RoboDK station: ALTERNATIVA 3 - PYTHON.rdk

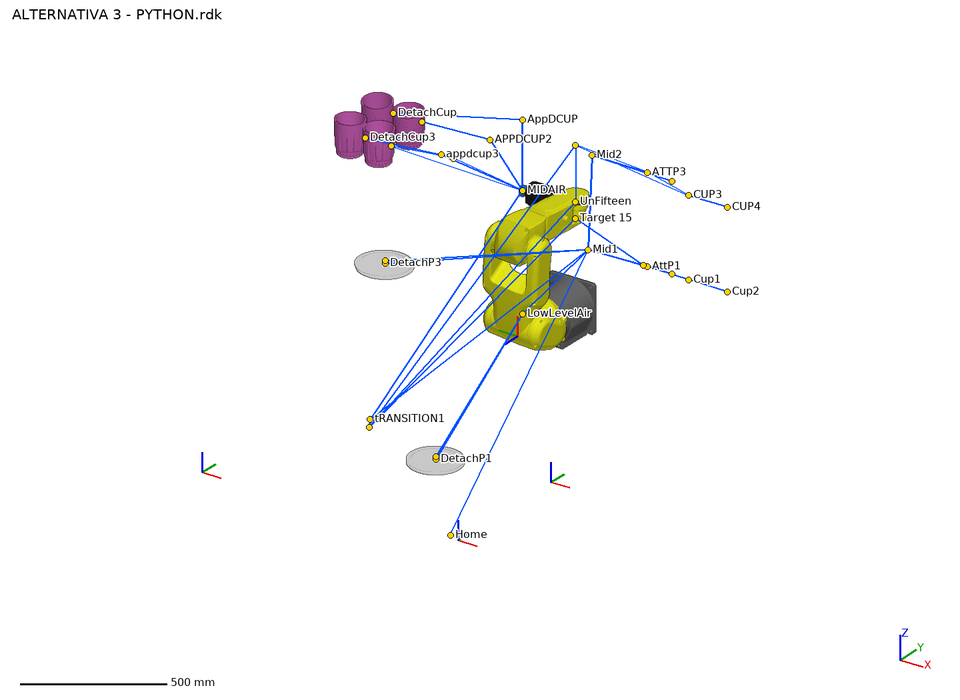
[picture v0: the station drawn from its stored meshes, robots at their saved joint values, targets as dots, program paths as lines]
Station ALTERNATIVA 3 (saved by RoboDK 6.0.0). Poses are relative to the parent item; angles as X-Y-Z fixed-axis rotations.
  - frame MUEBLE  at (-14.91, -46.19, 5.82) mm
    - object design2_refined_v2_without_doors at (0, 0, 0) mm, geometry from design2_refined_v2_without_doors.obj
      - item type 7 design2_refined_v2_without_doors-0
      - item type 7 design2_refined_v2_without_doors-1
      - item type 7 design2_refined_v2_without_doors-2
      - item type 7 design2_refined_v2_without_doors-3
      - item type 7 design2_refined_v2_without_doors-4
      - item type 7 design2_refined_v2_without_doors-5
      - item type 7 design2_refined_v2_without_doors-6
      - item type 7 design2_refined_v2_without_doors-7
      - item type 7 design2_refined_v2_without_doors-8
      - item type 7 design2_refined_v2_without_doors-9
      - item type 7 design2_refined_v2_without_doors-10
      - item type 7 design2_refined_v2_without_doors-11
      - item type 7 design2_refined_v2_without_doors-12
      - item type 7 design2_refined_v2_without_doors-13
      - item type 7 design2_refined_v2_without_doors-14
      - item type 7 design2_refined_v2_without_doors-15
      - item type 7 design2_refined_v2_without_doors-16
      - item type 7 design2_refined_v2_without_doors-17
      - item type 7 design2_refined_v2_without_doors-18
      - item type 7 design2_refined_v2_without_doors-19
      - item type 7 design2_refined_v2_without_doors-20
      - item type 7 design2_refined_v2_without_doors-21
      - item type 7 design2_refined_v2_without_doors-22
      - item type 7 design2_refined_v2_without_doors-23
      - item type 7 design2_refined_v2_without_doors-24
      - item type 7 design2_refined_v2_without_doors-25
      - item type 7 design2_refined_v2_without_doors-26
      - item type 7 design2_refined_v2_without_doors-27
  - frame Frame 3 at (1040, 513.81, 40) mm
    - target Home (joint target) at (96.91, -735, 120.39) mm, rotated rx -180 ry 0 rz -90 deg; joints [0, 0, 0, 0, 0, 0, 603.9] of Fanuc LR Mate 200iD
    - target AttP1 (Cartesian target) at (573.22, -246.74, 1075.18) mm, rotated rx -90.73 ry 0 rz -90 deg; joints [-34.498, 53.957, -76.428, 123.024, -82.505, -168.653, 603.9] of Fanuc LR Mate 200iD
    - target DetachP1 (Cartesian target) at (-411.21, -94.58, 10.61) mm, rotated rx 179.8 ry -0.07 rz 95.82 deg; joints [99.948, 86.361, -67, -98.991, -86.19, -16.417, 178.9] of Fanuc LR Mate 200iD
    - target AttP2 (Cartesian target) at (673.22, -246.74, 1075.18) mm, rotated rx -90.73 ry 0 rz -90 deg; joints [-44.12, 58.531, -67.298, 131.093, -74.625, -163.091, 603.9] of Fanuc LR Mate 200iD
    - target DetachP2 (Cartesian target) at (-411.21, -94.58, 20.61) mm, rotated rx 179.8 ry -0.07 rz 95.82 deg; joints [97.316, 86.024, -68.17, -96.585, -87.269, -15.858, 178.9] of Fanuc LR Mate 200iD
    - target ATTP3 (Cartesian target) at (573.19, -246.78, 1430.76) mm, rotated rx -90.72 ry 0 rz -90 deg; joints [-34.49, 53.95, -76.42, 123.02, -82.5, -168.65, 959.42] of Fanuc LR Mate 200iD
    - target Mid2 (Cartesian target) at (343.18, -246.78, 1430.76) mm, rotated rx -90.72 ry 0 rz -90 deg; joints [-2.136, 50.494, -87.492, 91.411, -89.937, -177.497, 959.42] of Fanuc LR Mate 200iD
    - target Mid1 (Cartesian target) at (333.22, -256.74, 1075.18) mm, rotated rx -90.73 ry 0 rz -90 deg; joints [-0.524, 48.486, -86.246, 89.797, -90.013, -176.246, 603.9] of Fanuc LR Mate 200iD
    - target DetachP3 (Cartesian target) at (-411.21, -394.58, 870.61) mm, rotated rx 179.8 ry -0.07 rz 95.82 deg; joints [56.153, 59.68, -30.838, -70.815, -118.669, -48.367, 603.9] of Fanuc LR Mate 200iD
    - target DetachP4 (Cartesian target) at (-411.21, -394.58, 880.61) mm, rotated rx 179.8 ry -0.07 rz 95.82 deg; joints [55.416, 60.777, -29.814, -70.867, -119.606, -49.236, 603.9] of Fanuc LR Mate 200iD
    - target AttachP4 (Cartesian target) at (673.25, -246.76, 1425.85) mm, rotated rx -90.73 ry 0.01 rz -90 deg; joints [-44.12, 58.53, -67.29, 131.09, -74.62, -163.09, 954.55] of Fanuc LR Mate 200iD
    - target Cup1 (Cartesian target) at (749.85, -254.56, 1076.96) mm, rotated rx -90.74 ry 0.07 rz -84.93 deg; joints [76.368, -58.415, 227.236, 18.8, -43.597, 167.309, 1061.69] of Fanuc LR Mate 200iD
    - target Target 13 (joint target) at (571.74, -270.38, 1089.27) mm, rotated rx -90.74 ry 0.07 rz -84.93 deg; joints [102.838, -41.717, 250.434, -14.839, -65.946, 184.939, 916.69] of Fanuc LR Mate 200iD
    - target Target 15 (joint target) at (290.04, -270.38, 1186.54) mm, rotated rx -36.26 ry -4.09 rz -87 deg; joints [170, -42.77, 247.74, -28.94, -65.13, 190.6, 633.12] of Fanuc LR Mate 200iD
    - target tRANSITION1 (Cartesian target) at (120, -1245, 768.12) mm, rotated rx 90 ry -8.75 rz 0 deg; joints [0, 0, 90, 0, 0, 261.25, 633.12] of Fanuc LR Mate 200iD
    - target Transition2 (Cartesian target) at (117.4, -1245, 738.35) mm, rotated rx -90 ry -1.24 rz 180 deg; joints [170, 0, 90, 0, 0, 261.24, 633.12] of Fanuc LR Mate 200iD
    - target DetachCup (Cartesian target) at (-508.51, -210.98, 1338.54) mm, rotated rx -88.72 ry -5.92 rz 93.84 deg; joints [51.581, 69.776, -64.617, -141.164, -73.844, -9.801, 881.49] of Fanuc LR Mate 200iD
    - target Cup2 (Cartesian target) at (909.85, -254.56, 1076.96) mm, rotated rx -90.74 ry 0.07 rz -84.93 deg; joints [80.035, -84.414, 196.552, 39.263, -14.612, 142.479, 1061.69] of Fanuc LR Mate 200iD
    - target DetachCup2 (Cartesian target) at (-388.51, -210.98, 1338.54) mm, rotated rx -88.72 ry -5.92 rz 93.84 deg; joints [41.981, 63.458, -78.354, -133.255, -85.98, -2.644, 881.49] of Fanuc LR Mate 200iD
    - target MIDAIR (Cartesian target) at (-57.84, -88.3, 1122.76) mm, rotated rx -88.72 ry -5.92 rz 93.83 deg; joints [-4.7, 82.95, -94.56, -86.27, -93.68, 10.39, 613.64] of Fanuc LR Mate 200iD
    - target AppDCUP (Cartesian target) at (-57.82, -88.33, 1390.6) mm, rotated rx -88.72 ry -5.92 rz 93.84 deg; joints [-4.703, 82.952, -94.565, -86.271, -93.69, 10.397, 881.49] of Fanuc LR Mate 200iD
    - target APPDCUP2 (Cartesian target) at (-57.82, -278.33, 1390.6) mm, rotated rx -88.72 ry -5.92 rz 93.84 deg; joints [-4.703, 48.487, -80.708, -87.263, -94.476, -3.473, 881.49] of Fanuc LR Mate 200iD
    - target CUP3 (Cartesian target) at (749.85, -254.56, 1396.96) mm, rotated rx -90.74 ry 0.07 rz -84.93 deg; joints [90.406, -57.172, 228.993, -1.647, -43.93, 181.084, 1276.69] of Fanuc LR Mate 200iD
    - target FIFteen (joint target) at (290.12, -270.38, 1464.1) mm, rotated rx -36.27 ry -4.09 rz -87 deg; joints [169.99, -42.77, 247.74, -28.94, -65.13, 190.6, 910.71] of Fanuc LR Mate 200iD
    - target DetachCup3 (Cartesian target) at (-498.51, -390.98, 1318.54) mm, rotated rx -90 ry 0 rz 90 deg; joints [52.184, 41.354, -48.276, -133.88, -58.279, -28.667, 881.49] of Fanuc LR Mate 200iD
    - target appdcup3 (Cartesian target) at (-188.51, -380.98, 1338.54) mm, rotated rx -88.72 ry -5.92 rz 93.84 deg; joints [16.598, 25.94, -69.048, -108.124, -87.435, -14.087, 881.49] of Fanuc LR Mate 200iD
    - target CUP4 (Cartesian target) at (909.85, -254.56, 1396.96) mm, rotated rx -90.74 ry 0.07 rz -84.93 deg; joints [-89.706, 63.915, -51.886, 178.586, -46.82, -179.124, 1276.69] of Fanuc LR Mate 200iD
    - target DetachCup4 (Cartesian target) at (-388.51, -390.98, 1318.54) mm, rotated rx -90 ry 0 rz 90 deg; joints [43.275, 31.43, -56.653, -128.185, -67.863, -25.6, 881.49] of Fanuc LR Mate 200iD
    - target APPDCUP4 (Cartesian target) at (-138.51, -380.98, 1338.54) mm, rotated rx -88.72 ry -5.92 rz 93.84 deg; joints [8.398, 24.874, -70.055, -100.444, -90.456, -13.82, 881.49] of Fanuc LR Mate 200iD
    - target wili (Cartesian target) at (573.19, -246.78, 1430.76) mm, rotated rx -90.72 ry 0 rz -90 deg; joints [145.51, -61.818, 229.982, -62.886, -69.058, 214.91, 959.42] of Fanuc LR Mate 200iD
    - target UnFifteen (joint target) at (290.12, -270.38, 1249.82) mm, rotated rx -36.27 ry -4.09 rz -87 deg; joints [169.99, -42.77, 247.74, -28.94, -65.13, 190.6, 696.43] of Fanuc LR Mate 200iD
    - target LowLevelAir (Cartesian target) at (-57.84, -88.36, 655.18) mm, rotated rx -88.73 ry -5.9 rz 93.84 deg; joints [-4.7, 82.94, -94.56, -86.26, -93.68, 10.38, 146.1] of Fanuc LR Mate 200iD
    - object PLATO3 at (-409.79, -107.42, 3.82) mm, rotated rx -0.53 ry 0.07 rz -84.18 deg, size 200 x 200 x 4 mm, geometry from tinker.obj
    - object PLATO4 at (-409.78, -107.42, 13.82) mm, rotated rx -0.53 ry 0.07 rz -84.18 deg, size 200 x 200 x 4 mm, geometry from tinker.obj
    - object PLATO1 at (-409.2, -407.4, 863.77) mm, rotated rx -0.53 ry 0.08 rz -84.17 deg, size 200 x 200 x 4 mm, geometry from tinker.obj
    - object PLATO2 at (-414.08, -407.88, 873.88) mm, rotated rx -0.53 ry 0.07 rz -84.17 deg, size 200 x 200 x 4 mm, geometry from tinker.obj
    - object VASO_3 at (-573.35, -220.21, 1237.76) mm, rotated rx 87.46 ry 5.78 rz -91.26 deg, size 110.6 x 132.4 x 110.6 mm, geometry from glass-obj.obj
    - object VASO_4 at (-443.36, -220.39, 1237.32) mm, rotated rx 87.46 ry 5.78 rz -91.26 deg, size 110.6 x 132.4 x 110.6 mm, geometry from glass-obj.obj
    - object VASO_1 at (-561.25, -406.24, 1242.36) mm, rotated rx 89.26 ry 0 rz -95.07 deg, size 110.6 x 132.4 x 110.6 mm, geometry from glass-obj.obj
    - object VASO_2 at (-441.29, -407.12, 1242.23) mm, rotated rx 89.26 ry 0 rz -95.07 deg, size 110.6 x 132.4 x 110.6 mm, geometry from glass-obj.obj
  - frame My Mechanism Base at (1040, -36.19, 40) mm
    - robot My Mechanism: 1 axes
        modified DH rows (alpha deg, a mm, theta deg, d mm): 0, 0, 0, 0 linear
        base shift (0, 0, 0) mm, rotated rx 180 ry 0 rz 180 deg
        joint limits [0] to [1500]; home [0]; saved at [613.64]
      - frame Fanuc LR Mate 200iD Base at (-120, 180, 120) mm, rotated rx -90 ry 0 rz -180 deg
        - robot Fanuc LR Mate 200iD: 6 axes, payload 7 kg, reach 717 mm, repeatability 0.02 mm, weight 25 kg
            modified DH rows (alpha deg, a mm, theta deg, d mm): 0, 0, 0, 330; -90, 50, -90, 0; 0, 330, 0, 0; -90, 35, 0, 335; 90, 0, 0, 0; -90, 0, 0, 80
            base shift (0, 0, -330) mm
            joint limits [-170, -100, -67, -190, -125, -360] to [170, 145, 213, 190, 124, 360]; home [0, 0, 0, 0, 0, 0]; saved at [-4.7, 82.95, -94.56, -86.27, -93.68, 10.39]
          - tool RobotiQ EPick Vacuum Gripper (1 Cup), TCP at (0, 0, 130) mm, size 75 x 83 x 136.1 mm
  - program Recall (1 instructions, listed below)
  - program Att (3 instructions, listed below)
  - program Det (1 instructions, listed below)
  - program Plates (103 instructions, listed below)
  - Python program Prog5 (listed below)
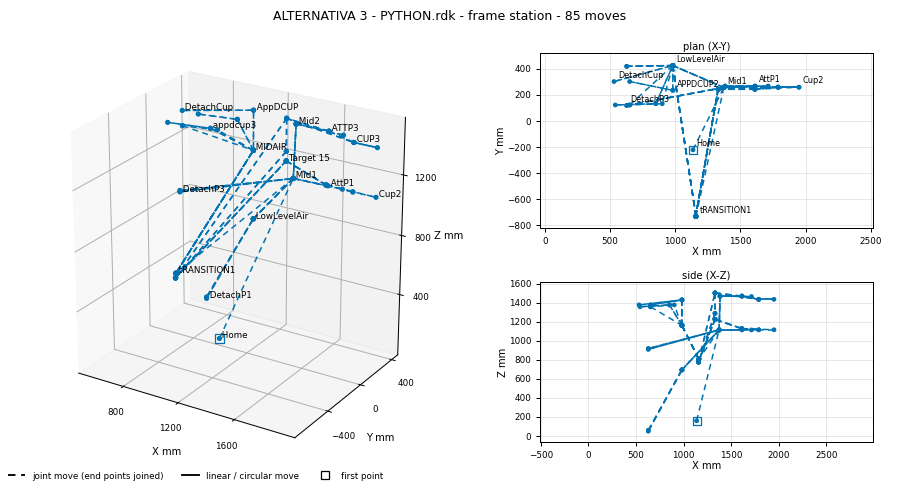
[picture p0: tool path of ALTERNATIVA 3 - PYTHON.rdk in frame station, 85 of 85 moves have a stored position in this frame; points joined in program order, loops and branches not executed]

--- program Recall (robot Fanuc LR Mate 200iD) ---
  Move objects

--- program Att (robot Fanuc LR Mate 200iD) ---
  Set Ref.: Frame 3
  Set Tool: RobotiQ EPick Vacuum Gripper (1 Cup)
  Attach to RobotiQ EPick Vacuum Gripper (1 Cup)

--- program Det (robot Fanuc LR Mate 200iD) ---
  Detach from RobotiQ EPick Vacuum Gripper (1 Cup)

--- program Plates (robot Fanuc LR Mate 200iD) ---
  Set Ref.: Frame 3
  Set Tool: RobotiQ EPick Vacuum Gripper (1 Cup)
  MoveJ (Home)
  MoveJ (Mid1)
  MoveJ (AttP1)
  Call Att
  MoveJ (Mid1)
  MoveJ (LowLevelAir)
  MoveJ (DetachP1)
  Call Det
  MoveJ (LowLevelAir)
  MoveJ (Mid1)
  MoveJ (AttP2)
  Call Att
  MoveJ (Mid1)
  MoveJ (LowLevelAir)
  MoveJ (DetachP2)
  Call Det
  MoveJ (LowLevelAir)
  MoveJ (Mid1)
  MoveJ (Mid2)
  MoveJ (ATTP3)
  Call Att
  MoveJ (Mid2)
  MoveJ (Mid1)
  MoveJ (DetachP3)
  Call Det
  MoveJ (Mid1)
  MoveJ (Mid2)
  MoveJ (AttachP4)
  Call Att
  MoveJ (Mid2)
  MoveJ (Mid1)
  MoveJ (DetachP4)
  Call Det
  MoveJ (Mid1)
  MoveJ (tRANSITION1)
  MoveJ (Transition2)
  MoveJ (Target 15)
  MoveJ (Target 13)
  MoveJ (Cup1)
  Call Att
  MoveJ (Target 13)
  MoveJ (Target 15)
  MoveJ (Transition2)
  MoveJ (tRANSITION1)
  MoveJ (MIDAIR)
  MoveJ (AppDCUP)
  MoveJ (DetachCup)
  Call Det
  MoveJ (AppDCUP)
  MoveJ (MIDAIR)
  MoveJ (tRANSITION1)
  MoveJ (Transition2)
  MoveJ (Target 15)
  MoveJ (Target 13)
  MoveJ (Cup2)
  Call Att
  MoveJ (Cup1)
  MoveJ (Target 13)
  MoveJ (Target 15)
  MoveJ (Transition2)
  MoveJ (tRANSITION1)
  MoveJ (MIDAIR)
  MoveJ (APPDCUP2)
  MoveJ (DetachCup2)
  Call Det
  MoveJ (APPDCUP2)
  MoveJ (MIDAIR)
  MoveJ (tRANSITION1)
  MoveJ (Transition2)
  MoveJ (FIFteen)
  MoveJ (CUP3)
  Call Att
  MoveJ (wili)
  MoveJ (FIFteen)
  MoveJ (UnFifteen)
  MoveJ (Transition2)
  MoveJ (tRANSITION1)
  MoveJ (MIDAIR)
  MoveJ (appdcup3)
  MoveJ (DetachCup3)
  Call Det
  MoveJ (appdcup3)
  MoveJ (MIDAIR)
  MoveJ (tRANSITION1)
  MoveJ (Transition2)
  MoveJ (FIFteen)
  MoveJ (CUP3)
  MoveL (CUP4)
  Call Att
  MoveL (CUP3)
  MoveJ (wili)
  MoveJ (FIFteen)
  MoveJ (UnFifteen)
  MoveJ (Transition2)
  MoveJ (tRANSITION1)
  MoveJ (MIDAIR)
  MoveJ (APPDCUP4)
  MoveJ (DetachCup4)
  Call Det
  MoveJ (DetachCup4)
  MoveJ (MIDAIR)

--- Python program Prog5 ---
# ============================================================
# ANALISIS ROBODK - PROGRAMA SIMPLE: Plates
#
# Datos mostrados:
# - Programa analizado
# - Tiempo ciclo
# - Distancia recorrida por el TCP en mm y m
# - Instrucciones válidas
# - Total de instrucciones
# - Total de movimientos
# - Nº MoveJ
# - Nº MoveL
# ============================================================

import os
import csv
import datetime

try:
    from robodk.robolink import *
except:
    from robolink import *


# ================= CONFIGURACIÓN =================

PROGRAMA = "Plates"
EXPORTAR_CSV = True


# ================= CONEXIÓN CON ROBODK =================

RDK = Robolink()

prog = RDK.Item(PROGRAMA, ITEM_TYPE_PROGRAM)

if not prog.Valid():
    RDK.ShowMessage("No se ha encontrado el programa: " + PROGRAMA)
    raise Exception("No se ha encontrado el programa: " + PROGRAMA)


# ================= DATOS DE TIEMPO Y DISTANCIA =================

try:
    resultado_update = prog.Update(COLLISION_ON, 3600)

    instrucciones_validas = int(resultado_update[0])
    tiempo_ciclo_s = float(resultado_update[1])
    distancia_tcp_mm = float(resultado_update[2])

except Exception as e:
    instrucciones_validas = 0
    tiempo_ciclo_s = 0.0
    distancia_tcp_mm = 0.0
    RDK.ShowMessage("Error al actualizar el programa: " + str(e))


distancia_tcp_m = distancia_tcp_mm / 1000.0


# ================= CONTAR MOVIMIENTOS =================

total_instrucciones = prog.InstructionCount()

total_movimientos = 0
num_movej = 0
num_movel = 0

for i in range(total_instrucciones):

    try:
        nombre, instype, movetype, es_target_articular, pose, joints = prog.Instruction(i)
    except:
        continue

    if instype == INS_TYPE_MOVE:

        total_movimientos += 1

        if movetype == MOVE_TYPE_JOINT:
            num_movej += 1

        elif movetype == MOVE_TYPE_LINEAR:
            num_movel += 1


# ================= MOSTRAR RESULTADOS =================

mensaje = ""
mensaje += "RESULTADOS DEL PROGRAMA ROBODK\n"
mensaje += "====================================\n\n"

mensaje += "Programa analizado: {}\n".format(prog.Name())
mensaje += "Tiempo ciclo: {:.3f} s\n".format(tiempo_ciclo_s)
mensaje += "Distancia recorrida por el TCP: {:.3f} mm\n".format(distancia_tcp_mm)
mensaje += "Distancia recorrida por el TCP: {:.3f} m\n".format(distancia_tcp_m)
mensaje += "Instrucciones válidas: {}\n".format(instrucciones_validas)
mensaje += "Total de instrucciones: {}\n".format(total_instrucciones)
mensaje += "Total de movimientos: {}\n".format(total_movimientos)
mensaje += "Nº MoveJ: {}\n".format(num_movej)
mensaje += "Nº MoveL: {}\n".format(num_movel)

print(mensaje)
RDK.ShowMessage(mensaje)


# ================= EXPORTAR A CSV =================

if EXPORTAR_CSV:

    escritorio = os.path.join(os.path.expanduser("~"), "Desktop")
    ruta_csv = os.path.join(escritorio, "resultados_robodk_Plates.csv")

    if not os.path.isdir(escritorio):
        ruta_csv = os.path.join(os.getcwd(), "resultados_robodk_Plates.csv")

    existe_archivo = os.path.isfile(ruta_csv)

    with open(ruta_csv, mode="a", newline="", encoding="utf-8-sig") as archivo:
        writer = csv.writer(archivo, delimiter=";")

        if not existe_archivo:
            writer.writerow([
                "Fecha",
                "Programa analizado",
                "Tiempo ciclo (s)",
                "Distancia TCP (mm)",
                "Distancia TCP (m)",
                "Instrucciones validas",
                "Total instrucciones",
                "Total movimientos",
                "MoveJ",
                "MoveL"
            ])

        writer.writerow([
            datetime.datetime.now().strftime("%Y-%m-%d %H:%M:%S"),
            prog.Name(),
            round(tiempo_ciclo_s, 3),
            round(distancia_tcp_mm, 3),
            round(distancia_tcp_m, 3),
            instrucciones_validas,
            total_instrucciones,
            total_movimientos,
            num_movej,
            num_movel
        ])

    print("\nCSV guardado en:")
    print(ruta_csv)
